FUNCTION ScaleAndRoundString : String
VAR_INPUT
	realValue 	: REAL;          // Die zu rundende REAL-Zahl
	scaleFactor : INT;           // Rundungsfaktor
END_VAR
VAR
END_VAR

ScaleAndRoundString := REAL_TO_STRING(INT_TO_REAL(REAL_TO_INT(realValue * scaleFactor)) / scaleFactor);

END_FUNCTION

(* stored: Version 1.1.0.1
   POU ScaleAndRoundString: Id {0262c68a-fc47-4aaf-bd89-714222ee8907}, SpecialFunc None *)
